# B&R Automation Studio project NAELD004C00R10L518F00 (part 29)

#### Act_Alarm.st - Do Not Change!!!
```iecst
(** 2019-03-25 **)
ACTION Act_Alarm:

	//Error
	IF EDGEPOS(eStatus = Error) THEN

		tyAlmData.sProgNm		:= p_sProgNm;
		tyAlmData.udiCode		:= udiStatus;
		tyAlmData.eSeverity		:= AlmSeverityError;
		tyAlmData.udiRunTime	:= tyAlmData.udiRunTime + 1;
		tyAlmData.bAlm			:= TRUE;
		tyAlmData.udiModuleNum  := udiModuleNum;
		g_sPneuExtSenProgNm		:= p_sProgNm;
		//Get Error Message
		IF tyAlmData.udiCode < 10000 OR tyAlmData.udiCode > 10099 THEN
			tyAlmData.sAlmMsg	:= 'Unknown';
			tyAlmData.sRcyMsg	:= 'Unknown';
		ELSE
			tyAlmData.sAlmMsg	:= a_tyAlmText[tyAlmData.udiCode].sAlmText;
			tyAlmData.sRcyMsg	:= a_tyAlmText[tyAlmData.udiCode].sRcyText;
		END_IF

		sStatTxt	:= tyAlmData.sAlmMsg;

	ELSIF bRstErr AND (tyAlmData.udiCode <> 0) THEN

		tyAlmData.udiCode	:= 0;
		tyAlmData.eSeverity	:= AlmSeverityNA;
		tyAlmData.sAlmMsg	:= '';
		tyAlmData.sRcyMsg	:= '';
		tyAlmData.bAlm			:= FALSE;
		sStatTxt	:= a_sStatText[eStat];

	END_IF

END_ACTION
```

#### Act_Background.st - Do Not Change!!!
```iecst
(** 2018-12-14 **)
ACTION Act_Background:

	IF p_bExtSen = FALSE THEN
		bExtended	:= FALSE;
	END_IF

END_ACTION
```

#### InputRef.var - Do Not Change!!!
```iecst
(*2019-03-25*)
(**)
(*General*)
VAR
	p_eAct : REFERENCE TO ePneuAction;
	p_udiRstErr : REFERENCE TO UDINT;
	p_bPrep : REFERENCE TO BOOL;
	p_bEn : REFERENCE TO BOOL;
	p_bDis : REFERENCE TO BOOL;
END_VAR
(**)
(*Configuration*)
VAR
	p_bManual : REFERENCE TO BOOL;
	p_bTwoCtrlIn : REFERENCE TO BOOL;
	p_bExtSafetySen : REFERENCE TO BOOL;
	p_bRetSafetySen : REFERENCE TO BOOL;
	p_sProgNm : REFERENCE TO STRING[15];
	p_tExtTO : REFERENCE TO TIME;
	p_tRetTO : REFERENCE TO TIME;
	p_bNtSettingsLoadDone : REFERENCE TO BOOL;
END_VAR
(**)
(*Input*)
VAR
	p_bExtSen : REFERENCE TO BOOL;
END_VAR
```

#### Local.var - Do Not Change!!!
```iecst
(*2019-04-30*)
(**)
(*Local Action, State & Status*)
VAR
	eAct : ePneuAction := PneuActIdle;
	eStat : ePneuAction := PneuActIdle;
	eStatus : eFBStatus := Idle;
	udiStatus : UDINT := 0;
	sStatTxt : STRING[200] := '';
	a_sStatText : ARRAY[0..50] OF STRING[200] := ['Idling','Set All','Reset All','Set Extend','Set Retract','Extending','Retracting','Retracting From Extend Sensor To Middle Sensor','Retracting From Middle Sensor To Retract Sensor','Extending From Retract Sensor To Middle Sensor','Extending From Middle Sensor To Extend Sensor',40('')];
END_VAR
(**)
(*Local Alarm*)
VAR
	tyAlmData : tyAlmDat;
	a_tyAlmText : ARRAY[10000..10099] OF tyAlmTxt := [(sAlmText:='Safety Check Error While Extending',sRcyText:='Safety System Has Been Triggered. All Operations Are Disable. Remove the Obstacle That Triggered The Safety Interlock To Resume Operation.'),(sAlmText:='Extend Sensor On Checking Time Out While Extending',sRcyText:='Sensor Timeout Expired Before Operation Completed. Sensor Operation Is Abnormal. Solve The Error To Resume Operation. '),(sAlmText:='Retract Sensor Off Checking Time Out While Extending',sRcyText:='Sensor Timeout Expired Before Operation Completed. Sensor Operation Is Abnormal. Solve The Error To Resume Operation.'),(sAlmText:='Safety Check Error While Retracting',sRcyText:='Safety System Has Been Triggered. All Operations Are Disable. Remove the Obstacle That Triggered The Safety Interlock To Resume Operation.'),(sAlmText:='Retract Sensor On Checking Time Out While Retracting',sRcyText:='Sensor Timeout Expired Before Operation Completed. Sensor Operation Is Abnormal. Solve The Error To Resume Operation.'),(sAlmText:='Extend Sensor Off Checking Time Out While Retracting',sRcyText:='Sensor Timeout Expired Before Operation Completed. Sensor Operation Is Abnormal. Solve The Error To Resume Operation.'),94((0))];
END_VAR
(**)
(*Local Output*)
VAR
	bExtCtrl : BOOL;
	bRetCtrl : BOOL;
	bTwoCtrlOut : BOOL := FALSE;
	bExtended : BOOL := FALSE;
	bRetracted : BOOL := FALSE;
END_VAR
(**)
(*Local Input*)
VAR
	udiRstErr : UDINT := 0;
	bPrep : BOOL := TRUE;
	bEn : BOOL := TRUE;
	bDis : BOOL := FALSE;
	bManual : BOOL := FALSE;
	bTwoCtrlIn : BOOL := FALSE;
	bExtSafetySen : BOOL := TRUE;
	bRetSafetySen : BOOL := TRUE;
	bExtSen : BOOL := FALSE;
	sProgNm : STRING[15] := 'TrolleyLck1';
	tExtTO : TIME := T#20s;
	tRetTO : TIME := T#20s;
	bNtSettingsLoadDone : BOOL := TRUE;
END_VAR
(**)
(*Local*)
VAR
	bRstErr : BOOL;
	udiRstErrOld : UDINT;
	bInitDone : BOOL;
	bInitialDone : BOOL;
	fbPneuExtChk : fbPneuExtSenExtChk;
	fbPneuRetChk : fbPneuExtSenRetChk;
	eStatOld : ePneuAction := PneuActIdle;
	udiModuleNum : UDINT := 2451;
END_VAR
```

### PneuExtSenTrolley2.var - Change By Project
```iecst
(*2019-03-25*)
(**)
(*Action & State & Status*)
VAR
	p_PneuExtSenTrlly2Stat : UDINT;
	p_PneuExtSenTrlly2Status : UDINT;
	p_PneuExtSenTrlly2StatTxt : UDINT;
END_VAR
(**)
(*Alarm*)
VAR
	p_PneuExtSenTrlly2AlmData : UDINT;
END_VAR
(**)
(*Output*)
VAR
	p_PneuExtSenTrlly2ExtCtrl : UDINT;
	p_PneuExtSenTrlly2RetCtrl : UDINT;
	p_PneuExtSenTrlly2TwoCtrlOut : UDINT;
	p_PneuExtSenTrlly2Extended : UDINT;
	p_PneuExtSenTrlly2Retracted : UDINT;
END_VAR
```

### Program Logical/Pneu/Trolley/PneuExtSenTrolley2 (IEC) - 1.00.0 - NtPneu v5.00.0

#### Local.var
```iecst
(*2019-04-30*)
(**)
(*Local Action, State & Status*)
VAR
	eAct : ePneuAction := PneuActIdle;
	eStat : ePneuAction := PneuActIdle;
	eStatus : eFBStatus := Idle;
	udiStatus : UDINT := 0;
	sStatTxt : STRING[200] := '';
	a_sStatText : ARRAY[0..50] OF STRING[200] := ['Idling','Set All','Reset All','Set Extend','Set Retract','Extending','Retracting','Retracting From Extend Sensor To Middle Sensor','Retracting From Middle Sensor To Retract Sensor','Extending From Retract Sensor To Middle Sensor','Extending From Middle Sensor To Extend Sensor',40('')];
END_VAR
(**)
(*Local Alarm*)
VAR
	tyAlmData : tyAlmDat;
	a_tyAlmText : ARRAY[10000..10099] OF tyAlmTxt := [(sAlmText:='Safety Check Error While Extending',sRcyText:='Safety System Has Been Triggered. All Operations Are Disable. Remove the Obstacle That Triggered The Safety Interlock To Resume Operation.'),(sAlmText:='Extend Sensor On Checking Time Out While Extending',sRcyText:='Sensor Timeout Expired Before Operation Completed. Sensor Operation Is Abnormal. Solve The Error To Resume Operation. '),(sAlmText:='Retract Sensor Off Checking Time Out While Extending',sRcyText:='Sensor Timeout Expired Before Operation Completed. Sensor Operation Is Abnormal. Solve The Error To Resume Operation.'),(sAlmText:='Safety Check Error While Retracting',sRcyText:='Safety System Has Been Triggered. All Operations Are Disable. Remove the Obstacle That Triggered The Safety Interlock To Resume Operation.'),(sAlmText:='Retract Sensor On Checking Time Out While Retracting',sRcyText:='Sensor Timeout Expired Before Operation Completed. Sensor Operation Is Abnormal. Solve The Error To Resume Operation.'),(sAlmText:='Extend Sensor Off Checking Time Out While Retracting',sRcyText:='Sensor Timeout Expired Before Operation Completed. Sensor Operation Is Abnormal. Solve The Error To Resume Operation.'),94((0))];
END_VAR
(**)
(*Local Output*)
VAR
	bExtCtrl : BOOL;
	bRetCtrl : BOOL;
	bTwoCtrlOut : BOOL := FALSE;
	bExtended : BOOL := FALSE;
	bRetracted : BOOL := FALSE;
END_VAR
(**)
(*Local Input*)
VAR
	udiRstErr : UDINT := 0;
	bPrep : BOOL := TRUE;
	bEn : BOOL := TRUE;
	bDis : BOOL := FALSE;
	bManual : BOOL := FALSE;
	bTwoCtrlIn : BOOL := FALSE;
	bExtSafetySen : BOOL := TRUE;
	bRetSafetySen : BOOL := TRUE;
	bExtSen : BOOL := FALSE;
	sProgNm : STRING[15] := 'TrolleyLck2';
	tExtTO : TIME := T#20s;
	tRetTO : TIME := T#20s;
	bNtSettingsLoadDone : BOOL := TRUE;
END_VAR
(**)
(*Local*)
VAR
	bRstErr : BOOL;
	udiRstErrOld : UDINT;
	bInitDone : BOOL;
	bInitialDone : BOOL;
	fbPneuExtChk : fbPneuExtSenExtChk;
	fbPneuRetChk : fbPneuExtSenRetChk;
	eStatOld : ePneuAction := PneuActIdle;
	udiModuleNum : UDINT := 2451;
END_VAR
```

#### Act_Alarm.st
```iecst
(** 2019-03-25 **)
ACTION Act_Alarm:

	//Error
	IF EDGEPOS(eStatus = Error) THEN

		tyAlmData.sProgNm		:= p_sProgNm;
		tyAlmData.udiCode		:= udiStatus;
		tyAlmData.eSeverity		:= AlmSeverityError;
		tyAlmData.udiRunTime	:= tyAlmData.udiRunTime + 1;
		tyAlmData.bAlm			:= TRUE;
		tyAlmData.udiModuleNum  := udiModuleNum;
		g_sPneuExtSenProgNm		:= p_sProgNm;		//snippet 15
		//Get Error Message
		IF tyAlmData.udiCode < 10000 OR tyAlmData.udiCode > 10099 THEN
			tyAlmData.sAlmMsg	:= 'Unknown';
			tyAlmData.sRcyMsg	:= 'Unknown';
		ELSE
			tyAlmData.sAlmMsg	:= a_tyAlmText[tyAlmData.udiCode].sAlmText;
			tyAlmData.sRcyMsg	:= a_tyAlmText[tyAlmData.udiCode].sRcyText;
		END_IF

		sStatTxt	:= tyAlmData.sAlmMsg;

	ELSIF bRstErr AND (tyAlmData.udiCode <> 0) THEN

		tyAlmData.udiCode	:= 0;
		tyAlmData.eSeverity	:= AlmSeverityNA;
		tyAlmData.sAlmMsg	:= '';
		tyAlmData.sRcyMsg	:= '';
		tyAlmData.bAlm			:= FALSE;
		sStatTxt	:= a_sStatText[eStat];

	END_IF

END_ACTION
```

#### Act_InitGlobal.st
```iecst
(** 2019-04-09 **)
ACTION Act_InitGlobal:

	(* Always Change If Project Change *)

	//Pass Data To Link
	p_bLinkOpsRun ACCESS p_OpsRun;
	p_bLinkDISafetyRlySig ACCESS p_DISafetyRlySig;

	//Pass Data To Internal Use
	p_bPrep ACCESS p_NtParamTrolleyLckPrep;
	p_bExtSen ACCESS p_DITrolleyExtRS2;
	p_tRetTO ACCESS p_NtParamTrolleyLckRetTO2;
	p_tExtTO ACCESS p_NtParamTrolleyLckExtTO2;
	p_bTwoCtrlIn ACCESS p_NtParamTrolleyLckTwoCtrlIn2;

	p_udiRstErr ACCESS p_RstErrReset;
	p_bManual ACCESS p_UIMnlMod;
	p_bNtSettingsLoadDone ACCESS p_StartupNtSettingsLoadDone;

	(* Always Change If Project Change *)

END_ACTION
```

#### Act_LinkAction.st
```iecst
(** 2019-04-09 **)
ACTION Act_LinkAction:

	IF p_bLinkOpsRun = TRUE THEN
		p_eAct ACCESS p_OpsMagConvLD2TrolleyLck;
	ELSIF p_bManual = TRUE THEN
		p_eAct ACCESS p_UITrolleyLckAct2;
	ELSE
		p_eAct ACCESS ADR(eAct);
	END_IF

END_ACTION
```

#### Act_Main.st
```iecst
(** 2019-01-10 **)
ACTION Act_Main:

	IF eStatOld <> eStat THEN
		fbPneuExtChk(bEn := FALSE);
		fbPneuRetChk(bEn := FALSE);

		sStatTxt	:= a_sStatText[eStat];

		eStatOld	:= eStat;

		eStatus		:= Busy;
	END_IF

	//Main
	CASE eStat OF

		PneuActIdle:
			eStatus	:= Idle;

		PneuActSetAll:
			IF eStatus = Idle OR eStatus = Busy THEN

				//Reset
				fbPneuExtChk(bEn := FALSE);
				fbPneuRetChk(bEn := FALSE);

				bExtCtrl	:= TRUE;
				bRetCtrl	:= TRUE;

				bRetracted	:= FALSE;

				eStatus	:= Done;

			END_IF

		PneuActRstAll:
			IF eStatus = Idle OR eStatus = Busy THEN

				//Reset
				fbPneuExtChk(bEn := FALSE);
				fbPneuRetChk(bEn := FALSE);

				bExtCtrl	:= FALSE;
				bRetCtrl	:= FALSE;

				bRetracted	:= FALSE;

				eStatus	:= Done;

			END_IF

		PneuActSetExt:
			IF eStatus = Idle OR eStatus = Busy THEN

				//Reset
				fbPneuExtChk(bEn := FALSE);
				fbPneuRetChk(bEn := FALSE);

				bExtCtrl	:= TRUE;
				bRetCtrl	:= FALSE;

				bExtended	:= TRUE;
				bRetracted	:= FALSE;

				eStatus	:= Done;

			END_IF

		PneuActSetRet:
			IF eStatus = Idle OR eStatus = Busy THEN

				//Reset
				fbPneuExtChk(bEn := FALSE);
				fbPneuRetChk(bEn := FALSE);

				bExtCtrl	:= FALSE;
				bRetCtrl	:= TRUE;

				bRetracted	:= TRUE;

				eStatus	:= Done;

			END_IF

		PneuActExt:
			IF eStatus = Idle OR eStatus = Busy THEN

				eStatus	:= Busy;

				//Reset
				fbPneuRetChk(bEn := FALSE);

				bExtCtrl	:= TRUE;
				bRetCtrl	:= FALSE;

				fbPneuExtChk.bExtSen	:= p_bExtSen;
				fbPneuExtChk.bExtSafety	:= p_bExtSafetySen;
				fbPneuExtChk(bEn := TRUE);

				IF fbPneuExtChk.udiStatus = 0 THEN
					bExtended	:= TRUE;
					bRetracted	:= FALSE;
					eStatus		:= Done;
				ELSIF fbPneuExtChk.udiStatus < 65534 THEN
					IF p_bTwoCtrlIn = TRUE THEN
						bExtCtrl	:= FALSE;
						bRetCtrl	:= FALSE;
					ELSE
						bExtCtrl	:= FALSE;
						bRetCtrl	:= TRUE;
					END_IF

					bRetracted	:= FALSE;

					eStatus		:= Error;

					IF fbPneuExtChk.udiStatus = 1507 THEN
						udiStatus	:= 10000;	//Safety Check Error While Extending
					ELSIF fbPneuExtChk.udiStatus = 1503 THEN
						udiStatus	:= 10001;	//Extend Sensor On Checking Time Out While Extending
					ELSE
						udiStatus	:= fbPneuExtChk.udiStatus;
					END_IF
				END_IF

			END_IF

		PneuActRet:
			IF eStatus = Idle OR eStatus = Busy THEN

				eStatus	:= Busy;

				//Reset
				fbPneuExtChk(bEn := FALSE);

				bExtCtrl	:= FALSE;
				bRetCtrl	:= TRUE;

				fbPneuRetChk.bExtSen	:= p_bExtSen;
				fbPneuRetChk.bRetSafety	:= p_bRetSafetySen;
				fbPneuRetChk(bEn := TRUE);

				IF fbPneuRetChk.udiStatus = 0 THEN
					bRetracted	:= TRUE;
					eStatus		:= Done;
				ELSIF fbPneuRetChk.udiStatus < 65534 THEN
					IF p_bTwoCtrlIn = TRUE THEN
						bExtCtrl	:= FALSE;
						bRetCtrl	:= FALSE;
					ELSE
						bExtCtrl	:= TRUE;
						bRetCtrl	:= FALSE;
					END_IF

					bRetracted	:= FALSE;

					eStatus		:= Error;

					IF fbPneuRetChk.udiStatus = 1508 THEN
						udiStatus	:= 10003;	//Safety Check Error While Retracting
					ELSIF fbPneuRetChk.udiStatus = 1504 THEN
						udiStatus	:= 10005;	//Extend Sensor Off Checking Time Out While Retracting
					ELSE
						udiStatus	:= fbPneuRetChk.udiStatus;
					END_IF
				END_IF

			END_IF

		ELSE
			IF eStatus = Idle OR eStatus = Busy THEN
				eStatus	:= Done;
			END_IF

	END_CASE

END_ACTION
```

#### Init.st
```iecst
(** 2019-03-25 **)
PROGRAM _INIT

	(* Always Change If Project Change *)

	//Pass Address To Global Address For External Use
	//Action, State & Status
	p_PneuExtSenTrlly2Stat			:= ADR(eStat);
	p_PneuExtSenTrlly2Status			:= ADR(eStatus);
	p_PneuExtSenTrlly2StatTxt		:= ADR(sStatTxt);

	//Alarm
	p_PneuExtSenTrlly2AlmData		:= ADR(tyAlmData);

	//Output
	p_PneuExtSenTrlly2ExtCtrl		:= ADR(bExtCtrl);
	p_PneuExtSenTrlly2RetCtrl		:= ADR(bRetCtrl);
	p_PneuExtSenTrlly2TwoCtrlOut	:= ADR(bTwoCtrlOut);
	p_PneuExtSenTrlly2Extended		:= ADR(bExtended);
	p_PneuExtSenTrlly2Retracted		:= ADR(bRetracted);

	(* Always Change If Project Change *)

END_PROGRAM
```

### Pneu2SenInShutter2.var - Change By Project
```iecst
(*2019-03-25*)
(**)
(*Action & State & Status*)
VAR
	p_Pneu2SenInShutterStat3 : UDINT;
	p_Pneu2SenInShutterStatus3 : UDINT;
	p_Pneu2SenInShutterStatTxt3 : UDINT;
END_VAR
(**)
(*Alarm*)
VAR
	p_Pneu2SenInShutterAlmData3 : UDINT;
END_VAR
(**)
(*Output*)
VAR
	p_Pneu2SenInShutterExtCtrl3 : UDINT;
	p_Pneu2SenInShutterRetCtrl3 : UDINT;
	p_Pneu2SenInShutterTwoCtrlOut3 : UDINT;
	p_Pneu2SenInShutterExtended3 : UDINT;
	p_Pneu2SenInShutterRetracted3 : UDINT;
END_VAR
```

### Program Logical/Pneu/Pneu2SenInShutter2 (IEC) - 1.00.0 - NtPneu v5.00.0

#### InputRef.var
```iecst
(*2019-03-25*)
(**)
(*General*)
VAR
	p_eAct : REFERENCE TO ePneuAction;
	p_udiRstErr : REFERENCE TO UDINT;
	p_bPrep : REFERENCE TO BOOL;
	p_bEn : REFERENCE TO BOOL;
	p_bDis : REFERENCE TO BOOL;
END_VAR
(**)
(*Configuration*)
VAR
	p_bSimu : REFERENCE TO BOOL;
	p_bManual : REFERENCE TO BOOL;
	p_bTwoCtrlIn : REFERENCE TO BOOL;
	p_bExtSafetySen : REFERENCE TO BOOL;
	p_bRetSafetySen : REFERENCE TO BOOL;
	p_sProgNm : REFERENCE TO STRING[15];
	p_tExtTO : REFERENCE TO TIME;
	p_tRetTO : REFERENCE TO TIME;
	p_bNtSettingsLoadDone : REFERENCE TO BOOL;
END_VAR
(**)
(*Input*)
VAR
	p_bExtSen : REFERENCE TO BOOL;
	p_bRetSen : REFERENCE TO BOOL;
END_VAR
```

#### InputRef_Link.var
```iecst
(*2019-04-09*)
(**)
(*External*)
VAR
	p_bLinkOpsRun : REFERENCE TO BOOL;
END_VAR
(**)
VAR
	p_bLinkDISafetyRlySig : REFERENCE TO BOOL;
	p_bLinkDIPullerRetRS : REFERENCE TO BOOL;
	p_bLinkDIConvLftSen : REFERENCE TO BOOL;
	p_bLinkProjShutter2Prep : REFERENCE TO BOOL;
	p_bLinkShutter1Extended : REFERENCE TO BOOL;
	p_bLinkShutter1Retracted : REFERENCE TO BOOL;
END_VAR
```

#### Local.var
```iecst
(*2019-04-30*)
(**)
(*Local Action, State & Status*)
VAR
	eAct : ePneuAction := PneuActIdle;
	eStat : ePneuAction := PneuActIdle;
	eStatus : eFBStatus := Idle;
	udiStatus : UDINT := 0;
	sStatTxt : STRING[200] := '';
	a_sStatText : ARRAY[0..50] OF STRING[200] := ['Idling','Set All','Reset All','Set Extend','Set Retract','Extending','Retracting','Retracting From Extend Sensor To Middle Sensor','Retracting From Middle Sensor To Retract Sensor','Extending From Retract Sensor To Middle Sensor','Extending From Middle Sensor To Extend Sensor',40('')];
END_VAR
(**)
(*Local Alarm*)
VAR
	tyAlmData : tyAlmDat;
	a_tyAlmText : ARRAY[10000..10099] OF tyAlmTxt := [(sAlmText:='Safety Check Error While Extending',sRcyText:='Safety System Has Been Triggered. All Operations Are Disable. Remove the Obstacle That Triggered The Safety Interlock To Resume Operation.'),(sAlmText:='Extend Sensor On Checking Time Out While Extending',sRcyText:='Sensor Timeout Expired Before Operation Completed. Sensor Operation Is Abnormal. Solve The Error To Resume Operation. '),(sAlmText:='Retract Sensor Off Checking Time Out While Extending',sRcyText:='Sensor Timeout Expired Before Operation Completed. Sensor Operation Is Abnormal. Solve The Error To Resume Operation.'),(sAlmText:='Safety Check Error While Retracting',sRcyText:='Safety System Has Been Triggered. All Operations Are Disable. Remove the Obstacle That Triggered The Safety Interlock To Resume Operation.'),(sAlmText:='Retract Sensor On Checking Time Out While Retracting',sRcyText:='Sensor Timeout Expired Before Operation Completed. Sensor Operation Is Abnormal. Solve The Error To Resume Operation.'),(sAlmText:='Extend Sensor Off Checking Time Out While Retracting',sRcyText:='Sensor Timeout Expired Before Operation Completed. Sensor Operation Is Abnormal. Solve The Error To Resume Operation.'),94((0))];
END_VAR
(**)
(*Local Output*)
VAR
	bExtCtrl : BOOL;
	bRetCtrl : BOOL;
	bTwoCtrlOut : BOOL := FALSE;
	bExtended : BOOL := FALSE;
	bRetracted : BOOL := FALSE;
END_VAR
(**)
(*Local Input*)
VAR
	udiRstErr : UDINT := 0;
	bPrep : BOOL := TRUE;
	bEn : BOOL := TRUE;
	bDis : BOOL := FALSE;
	bManual : BOOL := FALSE;
	bTwoCtrlIn : BOOL := FALSE;
	bExtSafetySen : BOOL := TRUE;
	bRetSafetySen : BOOL := TRUE;
	bExtSen : BOOL := FALSE;
	bRetSen : BOOL := FALSE;
	sProgNm : STRING[15] := 'Inlet Shutter2';
	tExtTO : TIME := T#20s;
	tRetTO : TIME := T#20s;
	bNtSettingsLoadDone : BOOL := TRUE;
END_VAR
(**)
(*Local*)
VAR
	bRstErr : BOOL;
	udiRstErrOld : UDINT;
	bInitDone : BOOL;
	bInitialDone : BOOL;
	fbPneuExtChk : fbPneuExtRetSenExtChk;
	fbPneuRetChk : fbPneuExtRetSenRetChk;
	eStatOld : ePneuAction := PneuActIdle;
	udiModuleNum : UDINT := 2551;
END_VAR
```

#### Act_InitGlobal.st
```iecst
(** 2019-04-09 **)
ACTION Act_InitGlobal:

	(* Always Change If Project Change *)

	//Pass Data To Link
	p_bLinkOpsRun ACCESS p_OpsRun;

	p_bLinkDISafetyRlySig ACCESS p_DISafetyRlySig;
	p_bLinkDIPullerRetRS ACCESS p_DIPullerRetRS;
	p_bLinkDIConvLftSen ACCESS p_DIConvLftSen;
	p_bLinkProjShutter2Prep ACCESS p_NtParamProjShutter2Prep;
	p_bLinkShutter1Extended ACCESS p_Pneu2SenInShutterExtended;
	p_bLinkShutter1Retracted ACCESS p_Pneu2SenInShutterRetracted;

	//Pass Data To Internal Use
	p_udiRstErr ACCESS p_RstErrReset;
	p_bPrep ACCESS p_NtParamProjInletShutPrep;
	p_bSimu ACCESS p_UISimuMod;
	p_bManual ACCESS p_UIMnlMod;
	p_bTwoCtrlIn ACCESS p_NtParamInShutterTwoCtrlIn;
//	p_sProgNm ACCESS p_NtParamInShutterProgNm;
	p_bExtSen ACCESS p_DIInShutterCloseRS2;
	p_bRetSen ACCESS p_DIInShutterOpenRS2;
	p_tExtTO ACCESS p_NtParamInShutterExtTO;
	p_tRetTO ACCESS p_NtParamInShutterRetTO;
	p_bNtSettingsLoadDone ACCESS p_StartupNtSettingsLoadDone;

	(* Always Change If Project Change *)

END_ACTION
```

#### Act_Link.st
```iecst
(** 2019-03-29 **)
ACTION Act_Link:

	p_bExtSafetySen	:= (p_bLinkDIPullerRetRS) AND (NOT p_bLinkDIConvLftSen);

//	p_bExtSafetySen	:= NOT p_bLinkDIConvLftSen;

	IF p_bLinkDISafetyRlySig = FALSE THEN
		bExtCtrl	:= FALSE;
		bRetCtrl	:= FALSE;
		bExtended	:= FALSE;
		bRetracted	:= FALSE;
	END_IF

END_ACTION
```

#### Act_LinkAction.st
```iecst
(** 2019-04-09 **)
ACTION Act_LinkAction:

	IF p_bLinkOpsRun = TRUE THEN
		p_eAct ACCESS p_OpsTravLifLDInletPneuAct2;
	ELSIF p_bManual = TRUE OR p_bSimu THEN
		p_eAct ACCESS p_UIInShutterAct2;
	ELSE
		p_eAct ACCESS ADR(eAct);
	END_IF

END_ACTION
```

#### Act_LinkEn.st
```iecst
(** 2019-01-11 **)
ACTION Act_LinkEn:

	//Link bPrep, bEn & bDis
	p_bEn ACCESS p_NtParamProjCurtainSenPrep;
	bDis := p_bLinkProjShutter2Prep = FALSE;

	IF p_bPrep AND p_bLinkProjShutter2Prep = FALSE THEN
		bExtended := p_bLinkShutter1Extended;
		bRetracted := p_bLinkShutter1Retracted;
		IF p_eAct <> PneuActIdle AND eStatus = Done THEN
			p_eAct := PneuActIdle;
		END_IF
	END_IF

END_ACTION
```

#### Init.st
```iecst
(** 2019-03-25 **)
PROGRAM _INIT

	(* Always Change If Project Change *)

	//Pass Address To Global Address For External Use
	//Action, State & Status
	p_Pneu2SenInShutterStat2		:= ADR(eStat);
	p_Pneu2SenInShutterStatus2		:= ADR(eStatus);
	p_Pneu2SenInShutterStatTxt2		:= ADR(sStatTxt);

	//Alarm
	p_Pneu2SenInShutterAlmData2		:= ADR(tyAlmData);

	//Output
	p_Pneu2SenInShutterExtCtrl2		:= ADR(bExtCtrl);
	p_Pneu2SenInShutterRetCtrl2		:= ADR(bRetCtrl);
	p_Pneu2SenInShutterTwoCtrlOut2	:= ADR(bTwoCtrlOut);
	p_Pneu2SenInShutterExtended2	:= ADR(bExtended);
	p_Pneu2SenInShutterRetracted2	:= ADR(bRetracted);

	(* Always Change If Project Change *)

END_PROGRAM
```

### Program Logical/Pneu/Pneu2SenInShutter3 (IEC) - 1.00.0 - NtPneu v5.00.0

#### InputRef_Link.var
```iecst
(*2019-04-09*)
(**)
(*External*)
VAR
	p_bLinkOpsRun : REFERENCE TO BOOL;
END_VAR
(**)
VAR
	p_bLinkDISafetyRlySig : REFERENCE TO BOOL;
	p_bLinkDIPullerRetRS : REFERENCE TO BOOL;
	p_bLinkDIConvLftSen : REFERENCE TO BOOL;
	p_bLinkProjShutter3Prep : REFERENCE TO BOOL;
	p_bLinkShutter1Extended : REFERENCE TO BOOL;
	p_bLinkShutter1Retracted : REFERENCE TO BOOL;
END_VAR
```

#### Local.var
```iecst
(*2019-04-30*)
(**)
(*Local Action, State & Status*)
VAR
	eAct : ePneuAction := PneuActIdle;
	eStat : ePneuAction := PneuActIdle;
	eStatus : eFBStatus := Idle;
	udiStatus : UDINT := 0;
	sStatTxt : STRING[200] := '';
	a_sStatText : ARRAY[0..50] OF STRING[200] := ['Idling','Set All','Reset All','Set Extend','Set Retract','Extending','Retracting','Retracting From Extend Sensor To Middle Sensor','Retracting From Middle Sensor To Retract Sensor','Extending From Retract Sensor To Middle Sensor','Extending From Middle Sensor To Extend Sensor',40('')];
END_VAR
(**)
(*Local Alarm*)
VAR
	tyAlmData : tyAlmDat;
	a_tyAlmText : ARRAY[10000..10099] OF tyAlmTxt := [(sAlmText:='Safety Check Error While Extending',sRcyText:='Safety System Has Been Triggered. All Operations Are Disable. Remove the Obstacle That Triggered The Safety Interlock To Resume Operation.'),(sAlmText:='Extend Sensor On Checking Time Out While Extending',sRcyText:='Sensor Timeout Expired Before Operation Completed. Sensor Operation Is Abnormal. Solve The Error To Resume Operation. '),(sAlmText:='Retract Sensor Off Checking Time Out While Extending',sRcyText:='Sensor Timeout Expired Before Operation Completed. Sensor Operation Is Abnormal. Solve The Error To Resume Operation.'),(sAlmText:='Safety Check Error While Retracting',sRcyText:='Safety System Has Been Triggered. All Operations Are Disable. Remove the Obstacle That Triggered The Safety Interlock To Resume Operation.'),(sAlmText:='Retract Sensor On Checking Time Out While Retracting',sRcyText:='Sensor Timeout Expired Before Operation Completed. Sensor Operation Is Abnormal. Solve The Error To Resume Operation.'),(sAlmText:='Extend Sensor Off Checking Time Out While Retracting',sRcyText:='Sensor Timeout Expired Before Operation Completed. Sensor Operation Is Abnormal. Solve The Error To Resume Operation.'),94((0))];
END_VAR
(**)
(*Local Output*)
VAR
	bExtCtrl : BOOL;
	bRetCtrl : BOOL;
	bTwoCtrlOut : BOOL := FALSE;
	bExtended : BOOL := FALSE;
	bRetracted : BOOL := FALSE;
END_VAR
(**)
(*Local Input*)
VAR
	udiRstErr : UDINT := 0;
	bPrep : BOOL := TRUE;
	bEn : BOOL := TRUE;
	bDis : BOOL := FALSE;
	bManual : BOOL := FALSE;
	bTwoCtrlIn : BOOL := FALSE;
	bExtSafetySen : BOOL := TRUE;
	bRetSafetySen : BOOL := TRUE;
	bExtSen : BOOL := FALSE;
	bRetSen : BOOL := FALSE;
	sProgNm : STRING[15] := 'Inlet Shutter3';
	tExtTO : TIME := T#20s;
	tRetTO : TIME := T#20s;
	bNtSettingsLoadDone : BOOL := TRUE;
END_VAR
(**)
(*Local*)
VAR
	bRstErr : BOOL;
	udiRstErrOld : UDINT;
	bInitDone : BOOL;
	bInitialDone : BOOL;
	fbPneuExtChk : fbPneuExtRetSenExtChk;
	fbPneuRetChk : fbPneuExtRetSenRetChk;
	eStatOld : ePneuAction := PneuActIdle;
	udiModuleNum : UDINT := 2551;
END_VAR
```

#### Act_InitGlobal.st
```iecst
(** 2019-04-09 **)
ACTION Act_InitGlobal:

	(* Always Change If Project Change *)

	//Pass Data To Link
	p_bLinkOpsRun ACCESS p_OpsRun;

	p_bLinkDISafetyRlySig ACCESS p_DISafetyRlySig;
	p_bLinkDIPullerRetRS ACCESS p_DIPullerRetRS;
	p_bLinkDIConvLftSen ACCESS p_DIConvLftSen;
	p_bLinkProjShutter3Prep ACCESS p_NtParamProjShutter3Prep;
	p_bLinkShutter1Extended ACCESS p_Pneu2SenInShutterExtended;
	p_bLinkShutter1Retracted ACCESS p_Pneu2SenInShutterRetracted;

	//Pass Data To Internal Use
	p_udiRstErr ACCESS p_RstErrReset;
	p_bPrep ACCESS p_NtParamProjInletShutPrep;
	p_bSimu ACCESS p_UISimuMod;
	p_bManual ACCESS p_UIMnlMod;
	p_bTwoCtrlIn ACCESS p_NtParamInShutterTwoCtrlIn;
//	p_sProgNm ACCESS p_NtParamInShutterProgNm;
	p_bExtSen ACCESS p_DIInShutterCloseRS3;
	p_bRetSen ACCESS p_DIInShutterOpenRS3;
	p_tExtTO ACCESS p_NtParamInShutterExtTO;
	p_tRetTO ACCESS p_NtParamInShutterRetTO;
	p_bNtSettingsLoadDone ACCESS p_StartupNtSettingsLoadDone;

	(* Always Change If Project Change *)

END_ACTION
```

#### Act_LinkAction.st
```iecst
(** 2019-04-09 **)
ACTION Act_LinkAction:

	IF p_bLinkOpsRun = TRUE THEN
		p_eAct ACCESS p_OpsTravLifLDInletPneuAct3;
	ELSIF p_bManual = TRUE OR p_bSimu THEN
		p_eAct ACCESS p_UIInShutterAct3;
	ELSE
		p_eAct ACCESS ADR(eAct);
	END_IF

END_ACTION
```

#### Act_LinkEn.st
```iecst
(** 2019-01-11 **)
ACTION Act_LinkEn:

	//Link bPrep, bEn & bDis
	p_bEn ACCESS p_NtParamProjCurtainSenPrep;
	bDis := p_bLinkProjShutter3Prep = FALSE;

	IF p_bPrep AND p_bLinkProjShutter3Prep = FALSE THEN
		bExtended := p_bLinkShutter1Extended;
		bRetracted := p_bLinkShutter1Retracted;
		IF p_eAct <> PneuActIdle AND eStatus = Done THEN
			p_eAct := PneuActIdle;
		END_IF
	END_IF

END_ACTION
```

#### Init.st
```iecst
(** 2019-03-25 **)
PROGRAM _INIT

	(* Always Change If Project Change *)

	//Pass Address To Global Address For External Use
	//Action, State & Status
	p_Pneu2SenInShutterStat3		:= ADR(eStat);
	p_Pneu2SenInShutterStatus3		:= ADR(eStatus);
	p_Pneu2SenInShutterStatTxt3		:= ADR(sStatTxt);

	//Alarm
	p_Pneu2SenInShutterAlmData3		:= ADR(tyAlmData);

	//Output
	p_Pneu2SenInShutterExtCtrl3		:= ADR(bExtCtrl);
	p_Pneu2SenInShutterRetCtrl3		:= ADR(bRetCtrl);
	p_Pneu2SenInShutterTwoCtrlOut3	:= ADR(bTwoCtrlOut);
	p_Pneu2SenInShutterExtended3	:= ADR(bExtended);
	p_Pneu2SenInShutterRetracted3	:= ADR(bRetracted);

	(* Always Change If Project Change *)

END_PROGRAM
```

### Pneu2SenOutShutter2.var - Change By Project
```iecst
(*2019-02-25*)
(**)
(*Action & State & Status*)
VAR
	p_Pneu2SenOutShutterStat2 : UDINT;
	p_Pneu2SenOutShutterStatus2 : UDINT;
	p_Pneu2SenOutShutterStatTxt2 : UDINT;
END_VAR
(**)
(*Alarm*)
VAR
	p_Pneu2SenOutShutterAlmData2 : UDINT;
END_VAR
(**)
(*Output*)
VAR
	p_Pneu2SenOutShutterExtCtrl2 : UDINT;
	p_Pneu2SenOutShutterRetCtrl2 : UDINT;
	p_Pneu2SenOutShutterTwoCtrlOut2 : UDINT;
	p_Pneu2SenOutShutterExtended2 : UDINT;
	p_Pneu2SenOutShutterRetracted2 : UDINT;
END_VAR
```

### Program Logical/Pneu/Pneu2SenOutShutter2 (IEC) - 1.00.0 - NtPneu v5.00.0

#### Local.var
```iecst
(*2019-04-30*)
(**)
(*Local Action, State & Status*)
VAR
	eAct : ePneuAction := PneuActIdle;
	eStat : ePneuAction := PneuActIdle;
	eStatus : eFBStatus := Idle;
	udiStatus : UDINT := 0;
	sStatTxt : STRING[200] := '';
	a_sStatText : ARRAY[0..50] OF STRING[200] := ['Idling','Set All','Reset All','Set Extend','Set Retract','Extending','Retracting','Retracting From Extend Sensor To Middle Sensor','Retracting From Middle Sensor To Retract Sensor','Extending From Retract Sensor To Middle Sensor','Extending From Middle Sensor To Extend Sensor',40('')];
END_VAR
(**)
(*Local Alarm*)
VAR
	tyAlmData : tyAlmDat;
	a_tyAlmText : ARRAY[10000..10099] OF tyAlmTxt := [(sAlmText:='Safety Check Error While Extending',sRcyText:='Safety System Has Been Triggered. All Operations Are Disable. Remove the Obstacle That Triggered The Safety Interlock To Resume Operation.'),(sAlmText:='Extend Sensor On Checking Time Out While Extending',sRcyText:='Sensor Timeout Expired Before Operation Completed. Sensor Operation Is Abnormal. Solve The Error To Resume Operation. '),(sAlmText:='Retract Sensor Off Checking Time Out While Extending',sRcyText:='Sensor Timeout Expired Before Operation Completed. Sensor Operation Is Abnormal. Solve The Error To Resume Operation.'),(sAlmText:='Safety Check Error While Retracting',sRcyText:='Safety System Has Been Triggered. All Operations Are Disable. Remove the Obstacle That Triggered The Safety Interlock To Resume Operation.'),(sAlmText:='Retract Sensor On Checking Time Out While Retracting',sRcyText:='Sensor Timeout Expired Before Operation Completed. Sensor Operation Is Abnormal. Solve The Error To Resume Operation.'),(sAlmText:='Extend Sensor Off Checking Time Out While Retracting',sRcyText:='Sensor Timeout Expired Before Operation Completed. Sensor Operation Is Abnormal. Solve The Error To Resume Operation.'),94((0))];
END_VAR
(**)
(*Local Output*)
VAR
	bExtCtrl : BOOL;
	bRetCtrl : BOOL;
	bTwoCtrlOut : BOOL := FALSE;
	bExtended : BOOL := FALSE;
	bRetracted : BOOL := FALSE;
END_VAR
(**)
(*Local Input*)
VAR
	udiRstErr : UDINT := 0;
	bPrep : BOOL := TRUE;
	bEn : BOOL := TRUE;
	bDis : BOOL := FALSE;
	p_bSimu : REFERENCE TO BOOL;
	bManual : BOOL := FALSE;
	bTwoCtrlIn : BOOL := FALSE;
	bExtSafetySen : BOOL := TRUE;
	bRetSafetySen : BOOL := TRUE;
	bExtSen : BOOL := FALSE;
	bRetSen : BOOL := FALSE;
	sProgNm : STRING[15] := 'OutShutter2';
	tExtTO : TIME := T#20s;
	tRetTO : TIME := T#20s;
	bNtSettingsLoadDone : BOOL := TRUE;
END_VAR
(**)
(*Local*)
VAR
	bRstErr : BOOL;
	udiRstErrOld : UDINT;
	bInitDone : BOOL;
	bInitialDone : BOOL;
	fbPneuExtChk : fbPneuExtRetSenExtChk;
	fbPneuRetChk : fbPneuExtRetSenRetChk;
	eStatOld : ePneuAction := PneuActIdle;
	udiModuleNum : UDINT := 2551;
END_VAR
```

#### Act_InitGlobal.st
```iecst
(** 2019-04-09 **)
ACTION Act_InitGlobal:

	(* Always Change If Project Change *)

	//Pass Data To Link
	p_bLinkOpsRun ACCESS p_OpsRun;

	p_bLinkDISafetyRlySig ACCESS p_DISafetyRlySig;
	p_bLinkInitOpsTravLifDone ACCESS p_OpsTravLifLDInitDone;
	p_bLinkMcParamOutShutDis ACCESS p_McParamOutShutterDis;
	p_bLinkDIConvClrSen ACCESS p_DIConvClrSen;

	//Pass Data To Internal Use
	p_udiRstErr ACCESS p_RstErrReset;
	p_bPrep ACCESS p_NtParamProjOutShutter2Prep;
//	p_bDis ACCESS p_McParamOutShutterDis;
	p_bSimu ACCESS p_UISimuMod;
	p_bManual ACCESS p_UIMnlMod;
	p_bTwoCtrlIn ACCESS p_NtParamOutShutterTwoCtrlIn;
//	p_sProgNm ACCESS p_NtParamOutShutterProgNm;
	p_bExtSen ACCESS p_DIOutShutterCloseRS2;
	p_bRetSen ACCESS p_DIOutShutterOpenRS2;
	p_tExtTO ACCESS p_NtParamOutShutterExtTO;
	p_tRetTO ACCESS p_NtParamOutShutterRetTO;
	p_bNtSettingsLoadDone ACCESS p_StartupNtSettingsLoadDone;

	(* Always Change If Project Change *)

END_ACTION
```

#### Act_Link.st
```iecst
(** 2019-03-29 **)
ACTION Act_Link:

	//p_bExtSafetySen := (p_bLinkDIConvClrSen = FALSE) ;

	IF p_bLinkDISafetyRlySig = FALSE THEN
		bExtCtrl	:= FALSE;
		bRetCtrl	:= FALSE;
		bExtended	:= FALSE;
		bRetracted	:= FALSE;
	END_IF

END_ACTION
```

#### Act_LinkAction.st
```iecst
(** 2019-04-09 **)
ACTION Act_LinkAction:

	IF p_bLinkOpsRun = TRUE THEN
		p_eAct ACCESS p_OpsTravLifLDOutletPneuAct2;
	ELSIF p_bManual = TRUE OR p_bSimu THEN
		p_eAct ACCESS p_UIOutShutterAct2;
	ELSE
		p_eAct ACCESS ADR(eAct);
	END_IF

END_ACTION
```

#### Act_LinkEn.st
```iecst
(** 2019-01-11 **)
ACTION Act_LinkEn:

	//Link bPrep, bEn & bDis
	IF p_bLinkOpsRun THEN
		p_bDis := p_bLinkMcParamOutShutDis AND p_bLinkInitOpsTravLifDone;
	ELSIF p_bManual THEN
		p_bDis	:= FALSE;
	END_IF

END_ACTION
```

#### Init.st
```iecst
(** 2019-03-25 **)
PROGRAM _INIT

	(* Always Change If Project Change *)

	//Pass Address To Global Address For External Use
	//Action, State & Status
	p_Pneu2SenOutShutterStat2		:= ADR(eStat);
	p_Pneu2SenOutShutterStatus2		:= ADR(eStatus);
	p_Pneu2SenOutShutterStatTxt2		:= ADR(sStatTxt);

	//Alarm
	p_Pneu2SenOutShutterAlmData2		:= ADR(tyAlmData);

	//Output
	p_Pneu2SenOutShutterExtCtrl2		:= ADR(bExtCtrl);
	p_Pneu2SenOutShutterRetCtrl2		:= ADR(bRetCtrl);
	p_Pneu2SenOutShutterTwoCtrlOut2	:= ADR(bTwoCtrlOut);
	p_Pneu2SenOutShutterExtended2	:= ADR(bExtended);
	p_Pneu2SenOutShutterRetracted2	:= ADR(bRetracted);

	(* Always Change If Project Change *)

END_PROGRAM
```

### Conv.typ - Change By Project
```iecst
(*2019-06-17*)
(**)
(*Action*)

TYPE
	eConvAction :
		(
		ConvActIdle,
		ConvActInit,
		ConvActInitRev,
		ConvActInitPshr,
		ConvActInitPuller,
		ConvActInitPuller1,
		ConvActInitRej,
		ConvActInitInsp,
		ConvActEnt,
		ConvActEntToInOff,
		ConvActEntRev,
		ConvActRev,
		ConvActRevImmedStart,
		ConvActEntPuller,
		ConvActEntRej,
		ConvActEntInsp,
		ConvActPreExit,
		ConvActRejResume,
		ConvActExit,
		ConvActExit1,
		ConvActExitPshr,
		ConvActExit1Pshr,
		ConvActPshrSetAll,
		ConvActPshrRstAll,
		ConvActPshrSetExt,
		ConvActPshrSetRet,
		ConvActPshrExt,
		ConvActPshrRet,
		ConvActPullerSetAll,
		ConvActPullerRstAll,
		ConvActPullerSetExt,
		ConvActPullerSetRet,
		ConvActPullerExt,
		ConvActPullerRet,
		ConvActRotSetAll,
		ConvActRotRstAll,
		ConvActRotSetHome,
		ConvActRotSetRmt,
		ConvActRotHome,
		ConvActRotRemote,
		ConvActRejSetAll,
		ConvActRejRstAll,
		ConvActRejSetUp,
		ConvActRejSetDown,
		ConvActRejUp,
		ConvActRejDown,
		ConvActStop,
		ConvActStopPshr,
		ConvActStopPuller,
		ConvActStopRej,
		ConvActSetMtrSigOnOrLToR,
		ConvActSetMtrDirOrRToL,
		ConvActRstMtrSigOnOrLToR,
		ConvActRstMtrDirOrRToL,
		ConvActSetMtrAll,
		ConvActRstMtrAll,
		ConvActEntPullerServo
		);
END_TYPE

(**)

TYPE
	eConvDir :
		(
		ConvDirLToR,
		ConvDirRToL,
		ConvDirLToL,
		ConvDirRToR
		);
END_TYPE
```

### PullConv.var - Change By Project
```iecst
(*2019-03-25*)
(**)
(*Action & State & Status*)
VAR
	p_PullConvStat : UDINT;
	p_PullConvStatus : UDINT;
	p_PullConvStatTxt : UDINT;
END_VAR
(**)
(*Alarm*)
VAR
	p_PullConvAlmData : UDINT;
END_VAR
(**)
(*Output*)
VAR
	p_PullConvHvBrd : UDINT;
	p_PullConvRejHvBrd : UDINT;
	p_PullConvInspHvBrd : UDINT;
	p_PullConvGdBrd : UDINT;
	p_PullConvLmtSenActivated : UDINT;
	p_PullConvMtrSigOnOrLToR : UDINT;
	p_PullConvMtrDirOrRToL : UDINT;
	p_PullConvPshrExtCtrl : UDINT;
	p_PullConvPshrTwoOutputControl : UDINT;
	p_PullConvPshrExtended : UDINT;
	p_PullConvPshrRetracted : UDINT;
	p_PullConvPullerExtCtrl : UDINT;
	p_PullConvPullerRetCtrl : UDINT;
	p_PullConvPullerTwoOutputControl : UDINT;
	p_PullConvPullerExtended : UDINT;
	p_PullConvPullerRetracted : UDINT;
	p_PullConvRotRemoteCtrl : UDINT;
	p_PullConvRotTwoOutputControl : UDINT;
	p_PullConvRotAtRemote : UDINT;
	p_PullConvRotAtHome : UDINT;
	p_PullConvRejectUpCtrl : UDINT;
	p_PullConvRejectDownCtrl : UDINT;
	p_PullConvRejectTwoOutputControl : UDINT;
	p_PullConvRejectAtUp : UDINT;
	p_PullConvRejectAtDown : UDINT;
END_VAR
```

### Program Logical/Conv/PullConv (IEC, version 1.00.0) - 1.00.0 - NtConv v5.00.0 , NtPneu v5.00.0

#### Init.st - Change By Project
```iecst
(** 2019-03-25 **)
PROGRAM _INIT

	(* Always Change If Project Change *)

	//Physical Configuration
	bGdBrdInit		:= TRUE;
	bGdBrdEnt		:= TRUE;
	diInitTm		:= 0;
	diTxInTimeOut	:= 60000;	//Greater Than Upstream SMEMA Transfer In Time Out

	//Pass Address To Global Address For External Use
	//Action, State & Status
	p_PullConvStat		:= ADR(eStat);
	p_PullConvStatus	:= ADR(eStatus);
	p_PullConvStatTxt	:= ADR(sStatTxt);

	//Alarm
	p_PullConvAlmData	:= ADR(tyAlmData);

	//Output
	p_PullConvHvBrd						:= ADR(bHvBrd);
	p_PullConvRejHvBrd					:= ADR(bRejHvBrd);
	p_PullConvInspHvBrd					:= ADR(bInspHvBrd);
	p_PullConvGdBrd						:= ADR(bGdBrd);
	p_PullConvLmtSenActivated			:= ADR(bLmtSenActivated);
	p_PullConvMtrSigOnOrLToR			:= ADR(bMtrSigOnOrLToR);
	p_PullConvMtrDirOrRToL				:= ADR(bMtrDirOrRToL);

	p_PullConvPshrExtCtrl				:= ADR(bPshrExtCtrl);
	p_PullConvPshrTwoOutputControl		:= ADR(bPshrTwoOutputControl);
	p_PullConvPshrExtended				:= ADR(bPshrExtended);
	p_PullConvPshrRetracted				:= ADR(bPshrRetracted);

	p_PullConvPullerExtCtrl				:= ADR(bPullerExtCtrl);
	p_PullConvPullerRetCtrl				:= ADR(bPullerRetCtrl);
	p_PullConvPullerTwoOutputControl	:= ADR(bPullerTwoOutputControl);
	p_PullConvPullerExtended			:= ADR(bPullerExtended);
	p_PullConvPullerRetracted			:= ADR(bPullerRetracted);

	p_PullConvRotRemoteCtrl				:= ADR(bRotRemoteCtrl);
	p_PullConvRotTwoOutputControl		:= ADR(bRotTwoOutputControl);
	p_PullConvRotAtRemote				:= ADR(bRotAtRemote);
	p_PullConvRotAtHome					:= ADR(bRotAtHome);

	p_PullConvRejectUpCtrl				:= ADR(bRejectUpCtrl);
	p_PullConvRejectDownCtrl			:= ADR(bRejectDownCtrl);
	p_PullConvRejectTwoOutputControl	:= ADR(bRejectTwoOutputControl);
	p_PullConvRejectAtUp				:= ADR(bRejectAtUp);
	p_PullConvRejectAtDown				:= ADR(bRejectAtDown);

	(* Always Change If Project Change *)

END_PROGRAM
```

#### Act_InitGlobal.st - Change By Project
```iecst
(** 2019-04-09 **)
ACTION Act_InitGlobal:

	(* Always Change If Project Change *)

	//Pass Data To Link
	p_bLinkOpsRun ACCESS p_OpsRun;

	p_bLinkUIBypsInitConv ACCESS p_UIOpsBypsInitConv;
	p_bLinkDISafetyRlySig ACCESS p_DISafetyRlySig;
	p_bLinkRotHomeSen ACCESS p_DIPullerRotHmRS;
	p_bLinkRotRemoteSen	ACCESS p_DIPullerRotRmRS;
	p_bLinkPullerExtSen ACCESS p_DIPullerExtRS;
	p_bLinkPullerRetSen ACCESS p_DIPullerRetRS;
	p_bLinkNtParamPullerRotPrep ACCESS p_NtParamProjPullerRotCylPrep;
	p_bSelfTest ACCESS p_DIMcSelfTest;
	p_bLinkDIRgtSen ACCESS p_DIConvRgtSen;
	p_bLinkOpsTravLifLDExitBrd ACCESS p_OpsTravLifLDExitBrd;
	p_bLinkDIPullerAntiJamSen ACCESS p_DIPullerAntiJamSen;
	p_bLinkPPTurnToHm ACCESS p_PPTurnToHm;

	//Pass Data To Internal Use
	p_udiRstErr ACCESS p_RstErrReset;
	p_bManual ACCESS p_UIMnlMod;
	p_bOnDirMod ACCESS p_NtParamPullConvOnDirMod;
	p_diInitTm ACCESS p_McParamConvInitTm;
	p_tMtrOffDlyTm ACCESS p_NtParamPullConvMtrOffDlyTm;
	p_diTxOutTimeOut ACCESS p_McParamTranOutErrDlyTm;
	p_eDirection ACCESS p_NtParamProjConvDir;
	p_sProgNm ACCESS p_NtParamPullConvProgNm;
	p_tPullerExtTO ACCESS p_NtParamPullConvPullExtTO;
	p_tPullerRetTO ACCESS p_NtParamPullConvPullRetTO;
	p_tRotHomeTO ACCESS p_NtParamPullConvRotHomeTO;
	p_tRotRemoteTO ACCESS p_NtParamPullConvRotRemoteTO;
	p_bLeftSen ACCESS p_DIConvLftSen;

	p_bNtSettingsLoadDone ACCESS p_StartupNtSettingsLoadDone;

	(* Always Change If Project Change *)

END_ACTION
```

#### InputRef_Link.var - Change By Project
```iecst
(*2019-04-09*)
(**)
(*External Data*)
VAR
	p_bLinkOpsRun : REFERENCE TO BOOL;
END_VAR
(**)
VAR
	p_bLinkUIBypsInitConv : REFERENCE TO BOOL;
	p_bLinkDISafetyRlySig : REFERENCE TO BOOL;
	p_bLinkRotHomeSen : REFERENCE TO BOOL;
	p_bLinkRotRemoteSen : REFERENCE TO BOOL;
	p_bLinkPullerExtSen : REFERENCE TO BOOL;
	p_bLinkPullerRetSen : REFERENCE TO BOOL;
	p_bLinkNtParamPullerRotPrep : REFERENCE TO BOOL;
	p_bSelfTest : REFERENCE TO BOOL;
	p_bLinkDIRgtSen : REFERENCE TO BOOL;
	p_bLinkOpsTravLifLDExitBrd : REFERENCE TO BOOL;
	p_bLinkDIPullerAntiJamSen : REFERENCE TO BOOL;
	p_bLinkPPTurnToHm : REFERENCE TO BOOL;
END_VAR
```

#### Act_LinkAction.st - Change By Project
```iecst
(** 2019-04-09 **)
ACTION Act_LinkAction:

	IF p_bLinkOpsRun = TRUE THEN
		p_eAct ACCESS p_OpsTravLifLDConvAct;
	ELSIF p_bManual = TRUE THEN
		p_eAct ACCESS p_UIPullConvAct;
	ELSE
		p_eAct ACCESS ADR(eAct);
		IF p_bLinkPPTurnToHm THEN
			p_eAct := ConvActRotHome;
		END_IF
		IF eStat = ConvActRotHome AND eStatus = Done THEN
			p_eAct := ConvActIdle;
			p_bLinkPPTurnToHm := FALSE ; //bi-dir
		END_IF

	END_IF

END_ACTION
```

#### Act_Link.st - Change By Project
```iecst
(** 2019-03-29 **)
ACTION Act_Link:

	IF p_bLinkDISafetyRlySig = FALSE THEN
		bPshrExtCtrl		:= FALSE;
		bPshrExtended		:= FALSE;
		bPshrRetracted		:= FALSE;

		bPullerExtCtrl		:= FALSE;
		bPullerRetCtrl		:= FALSE;
		bPullerExtended		:= FALSE;
		bPullerRetracted	:= FALSE;

		bRotRemoteCtrl		:= FALSE;
		bRotAtRemote		:= FALSE;
		bRotAtHome			:= FALSE;

		bRejectUpCtrl		:= FALSE;
		bRejectDownCtrl		:= FALSE;
		bRejectAtUp			:= FALSE;
		bRejectAtDown		:= FALSE;
	END_IF

	//Bypass Intializing Conveyor
	IF p_bLinkUIBypsInitConv THEN
		p_diInitTm ACCESS ADR(diInitTm);
	ELSE
		p_diInitTm ACCESS p_McParamConvInitTm;
	END_IF

	fbRightSenTm(IN:= bMtrSigOnOrLToR AND p_bRightSen = FALSE AND p_bLinkOpsTravLifLDExitBrd = FALSE, PT:= DINT_TO_TIME(p_diInitTm - 1000));
	fbRightSenTmOff(IN:= p_bLinkOpsTravLifLDExitBrd AND p_bRightSen, PT:= DINT_TO_TIME(p_diInitTm - 1000));
	IF p_bSelfTest = FALSE THEN
		p_bRightSen := p_bLinkDIRgtSen;
		fbBoardOffTm(IN:= p_bLeftSen = FALSE AND p_bRightSen = FALSE AND bMtrDirOrRToL = FALSE AND bMtrSigOnOrLToR = FALSE);
		IF EDGEPOS(fbBoardOffTm.Q) THEN
			bHvBrd := FALSE;
		END_IF
	ELSE
		IF fbRightSenTm.Q THEN
			p_bRightSen := TRUE;
			bHvBrd := TRUE;
		ELSIF fbRightSenTmOff.Q THEN
			p_bRightSen := FALSE;
			bHvBrd := FALSE;
		END_IF
	END_IF

	IF p_bLinkNtParamPullerRotPrep THEN
		p_bRotHomeSen := p_bLinkRotHomeSen;
		p_bRotRemoteSen := p_bLinkRotRemoteSen;
		p_bPullerRetSen := p_bLinkPullerRetSen;
		p_bPullerExtSen := p_bLinkPullerExtSen;
	ELSE
		p_bRotHomeSen := bRotRemoteCtrl = FALSE;
		p_bRotRemoteSen := bRotRemoteCtrl;
		p_bPullerRetSen := p_bLinkPullerRetSen;
		p_bPullerExtSen := p_bLinkPullerExtSen;
	END_IF

	//Antijam alm , hold pos
	IF (p_bLinkOpsRun = FALSE OR bPullerRetCtrl) AND p_bLinkDIPullerAntiJamSen = FALSE THEN
		eStatus := Error;
		udiStatus := 10125; //'Puller AntiJam Sensor On'
		bPullerRetCtrl		:= FALSE;
		bMtrSigOnOrLToR		:= FALSE;
	END_IF

END_ACTION
```
